(* IEC 61131-3 sources: ICS_Water_testbed/ics_sandbox/sim/physic_simulation, 6 files *)

(* ---- PLC1.st ---- *)
PROGRAM PLC1
  VAR
    P101_Q AT %QX0.0 : BOOL;
    P101_I AT %IX0.0 : BOOL;
    P102_Q AT %QX0.1 : BOOL;
    P102_I AT %IX0.1 : BOOL;
    FIT201_Q AT %QW0 : INT;
    FIT201_I AT %IW0 : INT;
    LIT101_Q AT %QW1 : INT;
    LIT101_I AT %IW1 : INT;
  END_VAR

  P101_Q := P101_I;
  P102_Q := P102_I;
  FIT201_Q := FIT201_I;
  LIT101_Q := LIT101_I;
END_PROGRAM

CONFIGURATION Config0

  RESOURCE Res0 ON PLC
    TASK task0(INTERVAL := T#20ms,PRIORITY := 0);
    PROGRAM instance0 WITH task0 : PLC1;
  END_RESOURCE
END_CONFIGURATION

(* ---- PLC2.st ---- *)
PROGRAM PLC2
  VAR
    MV201_Q AT %QX0.4 : BOOL;
    MV201_I AT %IX0.4 : BOOL;
  END_VAR

  MV201_Q := MV201_I;
END_PROGRAM

CONFIGURATION Config0

  RESOURCE Res0 ON PLC
    TASK task0(INTERVAL := T#20ms,PRIORITY := 0);
    PROGRAM instance0 WITH task0 : PLC2;
  END_RESOURCE
END_CONFIGURATION

(* ---- PLC3.st ---- *)
PROGRAM PLC3
  VAR
    P301_Q AT %QX0.5 : BOOL;
    P301_I AT %IX0.5 : BOOL;
    P302_Q AT %QX0.6 : BOOL;
    P302_I AT %IX0.6 : BOOL;
    MV302_Q AT %QX0.7 : BOOL;
    MV302_I AT %IX0.7 : BOOL;
    LIT301_Q AT %QW2 : INT;
    LIT301_I AT %IW2 : INT;
    FIT301_Q AT %QW3 : INT;
    FIT301_I AT %IW3 : INT;
  END_VAR

  P301_Q := P301_I;
  P302_Q := P302_I;
  MV302_Q := MV302_I;
  LIT301_Q := LIT301_I;
  FIT301_Q := FIT301_I;
END_PROGRAM

CONFIGURATION Config0

  RESOURCE Res0 ON PLC
    TASK task0(INTERVAL := T#20ms,PRIORITY := 0);
    PROGRAM instance0 WITH task0 : PLC3;
  END_RESOURCE
END_CONFIGURATION

(* ---- PLC4.st ---- *)
PROGRAM PLC4
  VAR
    P401_Q AT %QX1.0 : BOOL;
    P401_I AT %IX1.0 : BOOL;
    P402_Q AT %QX1.1 : BOOL;
    P402_I AT %IX1.1 : BOOL;
    LIT401_Q AT %QW4 : INT;
    LIT401_I AT %IW4 : INT;
    FIT401_Q AT %QW5 : INT;
    FIT401_I AT %IW5 : INT;
  END_VAR

  P401_Q := P401_I;
  P402_Q := P402_I;
  LIT401_Q := LIT401_I;
  FIT401_Q := FIT401_I;
END_PROGRAM

CONFIGURATION Config0

  RESOURCE Res0 ON PLC
    TASK task0(INTERVAL := T#20ms,PRIORITY := 0);
    PROGRAM instance0 WITH task0 : PLC4;
  END_RESOURCE
END_CONFIGURATION

(* ---- PLC5.st ---- *)
PROGRAM PLC5
  VAR
    MV501_Q AT %QX1.2 : BOOL;
    MV501_I AT %IX1.2 : BOOL;
    MV503_Q AT %QX1.3 : BOOL;
    MV503_I AT %IX1.3 : BOOL;
    P501_Q AT %QX1.4 : BOOL;
    P501_I AT %IX1.4 : BOOL;
    P502_Q AT %QX1.5 : BOOL;
    P502_I AT %IX1.5 : BOOL;
    FIT501_Q AT %QW6 : INT;
    FIT501_I AT %IW6 : INT;
    FIT502_Q AT %QW7 : INT;
    FIT502_I AT %IW7 : INT;
    FIT503_Q AT %QW8 : INT;
    FIT503_I AT %IW8 : INT;
  END_VAR

  MV501_Q := MV501_I;
  MV503_Q := MV503_I;
  P501_Q := P501_I;
  P502_Q := P502_I;
  FIT501_Q := FIT501_I;
  FIT502_Q := FIT502_I;
  FIT503_Q := FIT503_I;
END_PROGRAM

CONFIGURATION Config0

  RESOURCE Res0 ON PLC
    TASK task0(INTERVAL := T#20ms,PRIORITY := 0);
    PROGRAM instance0 WITH task0 : PLC5;
  END_RESOURCE
END_CONFIGURATION

(* ---- PLC6.st ---- *)
PROGRAM PLC6
  VAR
    P601_Q AT %QX1.6 : BOOL;
    P601_I AT %IX1.6 : BOOL;
    P603_Q AT %QX1.7 : BOOL;
    P603_I AT %IX1.7 : BOOL;
    LS601_Q AT %QW9 : INT;
    LS601_I AT %IW9 : INT;
    LS603_Q AT %QW10 : INT;
    LS603_I AT %IW10 : INT;
  END_VAR

  P601_Q := P601_I;
  P603_Q := P603_I;
  LS601_Q := LS601_I;
  LS603_Q := LS603_I;
END_PROGRAM

CONFIGURATION Config0

  RESOURCE Res0 ON PLC
    TASK task0(INTERVAL := T#20ms,PRIORITY := 0);
    PROGRAM instance0 WITH task0 : PLC6;
  END_RESOURCE
END_CONFIGURATION
